FUNCTION_BLOCK FB_eChillerSystem EXTENDS FB_SystemContinous
VAR_INPUT
	fExternalTemperature : REAL; //External temperature of buffer storage
END_VAR
VAR_OUTPUT
END_VAR
VAR
	//component - Efficient Energy eChiller 45-II
	eChiller : FB_eChiller;
	
	//component - valve 138
	ST_SV138DefaultParameters : ST_MixingValveDefaultParameters := (bFeedbackSignal := TRUE,aSetPointLimitsPosition := [0,100],fDefaultPosition := 0);
	SV138 : FB_MixingValve := (ST_DefaultParameters := ST_SV138DefaultParameters); //valve motor needs continous signal but operates only between extreme positions	
	
	//internal variables
	bSetStatusOn_eChiller : BOOL;
	bSetStatusOn_SV138 : BOOL;
END_VAR

MAIN();
eChiller(
	bSetStatusOnAutomatic := bSetStatusOn_eChiller,
	fSetPointAutomatic := fSetPoint,
	bAlgorithmPermission := bAlgorithmPermission,
	fExternalTemperature := fExternalTemperature);
eChiller.SetState();

//valve may only control position, not temperatures
SV138(
	bSetStatusOnAutomatic := bSetStatusOn_SV138,
	fSetPointAutomatic := 100,
	bAlgorithmPermission := bAlgorithmPermission,
	nControlModeAutomatic := 0);
SV138.SetState_AI_AO();

METHOD PROTECTED  CheckError : BOOL
VAR_INPUT
END_VAR
VAR
	bError_eChiller : BOOL := FALSE;
	bError_SV138 : BOOL := FALSE;
END_VAR
VAR_OUTPUT
	bError : BOOL := FALSE;
END_VAR
//Check chiller for error
bError_eChiller := eChiller.bError;

//Check valve SV138 for error
IF SV138.fOperatingPoint <= 95 AND eChiller.bStatusOn THEN
	bError_SV138 := TRUE;
END_IF

bError := bError_eChiller OR bError_SV138;
END_METHOD

METHOD PROTECTED  Operational : BOOL
VAR_INPUT
END_VAR
VAR_OUTPUT
	bSwitchToWorking : BOOL := FALSE;
END_VAR
bSetStatusOn_eChiller := TRUE;

//Wait until eChiller is switched on
IF eChiller.bStatusOn THEN
	bSwitchToWorking := TRUE;
END_IF
END_METHOD

METHOD PROTECTED  RampDown : BOOL
VAR_INPUT
END_VAR
VAR_OUTPUT
	bRampDownFinished : BOOL := FALSE;
END_VAR
bSetStatusOn_eChiller := FALSE;

//Wait until eChiller is switched off before closing valve
IF NOT eChiller.bStatusOn THEN
	bSetStatusOn_SV138 := FALSE;
END_IF

//Wait until valve is closed and ensure that eChiller is not switched on meanwhile
IF SV138.fOperatingPoint < 5 AND NOT eChiller.bStatusOn THEN
	bRampDownFinished := TRUE;
END_IF
END_METHOD

METHOD PROTECTED  RampUp : BOOL
VAR_INPUT
END_VAR
VAR_OUTPUT
	bRampUpFinished : BOOL := FALSE;
END_VAR
bSetStatusOn_SV138 := TRUE;

//Wait until valve is opened
IF SV138.fOperatingPoint > 95 THEN
	bRampUpFinished := TRUE;
END_IF
END_METHOD

METHOD PROTECTED SetSetPointLimits : BOOL
VAR_INPUT
END_VAR
aSetPointLimits[1] := eChiller.ST_DefaultParameters.aSetPointLimitsTemperature[1];
aSetPointLimits[2] := eChiller.ST_DefaultParameters.aSetPointLimitsTemperature[2];
END_METHOD

METHOD PROTECTED  Working : BOOL
VAR_INPUT
END_VAR
VAR_OUTPUT
	bSwitchToOperational : BOOL := FALSE;
END_VAR
//Check if eChiller is switched off (manually) but valve is still opened
IF NOT eChiller.bStatusOn AND SV138.fOperatingPoint > 95 THEN
	bSwitchToOperational := TRUE;
END_IF
END_METHOD

END_FUNCTION_BLOCK

(* stored: Version 1.1.0.1, ProductVersion 3.1.4024.9
   POU FB_eChillerSystem: Id {a7bd099c-d170-4645-8110-744e5a951345}, SpecialFunc None
   Method CheckError: Id {5f9e515c-f85f-4ce5-b9e9-0e4f29819e9c}
   Method Operational: Id {d9c42dcc-569b-4e06-be90-b76a61d09d20}
   Method RampDown: Id {6d7dce04-b763-4447-a5fc-f6af1df4542c}
   Method RampUp: Id {555d673f-1ed6-4f62-9777-be9332104160}
   Method SetSetPointLimits: Id {30aae5c2-589e-40f1-a55c-f3d4f4c0d944}
   Method Working: Id {f350f870-390c-44aa-8527-7f885801638b} *)
